PROGRAM NCI
VAR
  bInit                     : BOOL;
  eInit                     : E_PROGRESS;

  nChn,
  nChnInit,
  nAxis,
  nAxisInit                 : UINT;

  stMsg                     : ST_Message;

END_VAR

//-----------------------------------------------------------------------------------------------------------------
// check if compiler define is present [PLC_STATE_DRIVE/CompilerDefines/Manual: NCI]
// see PLC_CONSTANT for conditional pragma
//-----------------------------------------------------------------------------------------------------------------
IF NOT PLC_CONSTANT.NCI_ACTIVE THEN eInit   := E_PROGRESS.PROGRESS_NOT_EXIST; RETURN; END_IF
//-----------------------------------------------------------------------------------------------------------------
//-----------------------------------------------------------------------------------------------------------------
// check for MAIN.eInit
//-----------------------------------------------------------------------------------------------------------------
IF NOT (MAIN.eInit = E_PROGRESS.PROGRESS_DONE) THEN eInit   := E_PROGRESS.PROGRESS_INVALID; RETURN; END_IF
//-----------------------------------------------------------------------------------------------------------------
//-----------------------------------------------------------------------------------------------------------------
// /assign dataflow
//-----------------------------------------------------------------------------------------------------------------
FOR nChn := 1 TO MAX_NCI_CH
DO
  // NCI axis configuration --> NC AxisId used
  GVL_NCI.NciCtrl[nChn].ItfChannel.CfgAxes          := ADR(GVL_NCI.AxisConfig[nChn]);

  // R Parameter properties
  GVL_NCI.NciCtrl[nChn].ItfChannel.R_ParameterRead  := ADR(GVL_NCI.R_ParameterRead[nChn]);
  GVL_NCI.NciCtrl[nChn].ItfChannel.R_ParameterWrite := ADR(GVL_NCI.R_ParameterWrite[nChn]);

  // ProgName for channel
  GVL_NCI.NciCtrl[nChn].ItfChannel.Prog             := GVL_NCI.ChannelCtrl[nChn].sProgramName;

  // check REAL value to avoid exception
  IF NOT IsFinite(F_Real(GVL_NCI.ChannelCtrl[nChn].rOverride))
  THEN
    GVL_NCI.NciCtrl[nChn].ItfChannel.Override       := 0.0;
  ELSE
    GVL_NCI.NciCtrl[nChn].ItfChannel.Override       := GVL_NCI.ChannelCtrl[nChn].rOverride;
  END_IF

  // command and state structure assignement
  GVL_NCI.NciCtrl[nChn].ChnCtrl                     := ADR(GVL_NCI.ChannelCtrl[nChn]);
  GVL_NCI.NciCtrl[nChn].ChnState                    := ADR(GVL_NCI.ChannelState[nChn]);
END_FOR
//-----------------------------------------------------------------------------------------------------------------
// assign dataflow/
//-----------------------------------------------------------------------------------------------------------------
//-----------------------------------------------------------------------------------------------------------------
// /INIT
//-----------------------------------------------------------------------------------------------------------------
IF NOT bInit
THEN
  CASE eInit
  OF
    E_PROGRESS.PROGRESS_INVALID,
    E_PROGRESS.PROGRESS_DONE:
      FOR nChn := 1 TO MAX_NCI_CH
      DO
        GVL_MSG.MessageLevelNciChn[nChn]            := E_MessageType.eMessageVerbose;//GVL_MSG.MessageLevel;
      END_FOR
      nChnInit                                      := 1;
      eInit                                         := E_PROGRESS.PROGRESS_INIT;
    //-----------------------------------------------------------------------------
    //-----------------------------------------------------------------------------
    E_PROGRESS.PROGRESS_INIT:
      stMsg.eType                                   := E_MessageType.eMessageInfo;
      stMsg.eDevice                                 := e_Device.Device_Nci;
      stMsg.eSubdevice                              := e_SubDevice.MainInit;
      stMsg.iErrorNumber                            := MAX_AXIS;
      stMsg.sText                                   := concat('NCI.eInit: ', TO_STRING(eInit));
      f_MessageSet(stMsg);                          

      eInit                                         := E_PROGRESS.PROGRESS_BUSY;
    //-----------------------------------------------------------------------------
    //-----------------------------------------------------------------------------
    E_PROGRESS.PROGRESS_BUSY:
      eInit                                         := E_PROGRESS.PROGRESS_PREPARE;
    //-----------------------------------------------------------------------------
    //-----------------------------------------------------------------------------
    E_PROGRESS.PROGRESS_PREPARE:
      stMsg.eType                                   := E_MessageType.eMessageVerbose;
      stMsg.eDevice                                 := e_Device.Device_Nci;
      stMsg.eSubdevice                              := e_SubDevice.NciStartUp;
      stMsg.iErrorNumber                            := nChnInit;
      stMsg.sText                                   := concat('nChnInit: ', TO_STRING(nChnInit));

      IF (GVL_MSG.MessageLevelNciChn[nChnInit] = E_MessageType.eMessageVerbose)
      THEN
        f_MessageSet(stMsg);
      END_IF

      GVL_NCI.ChannelCtrl[nChnInit].eCmd            := E_NCI_CTRL.NULL;
      eInit                                         := E_PROGRESS.PROGRESS_STARTUP;
    //-----------------------------------------------------------------------------
    //-----------------------------------------------------------------------------
    E_PROGRESS.PROGRESS_STARTUP:
      GVL_NCI.ChannelCtrl[nChnInit].eCmd            := E_NCI_CTRL.INIT;

      IF (GVL_NCI.ChannelState[nChnInit].eState = E_NCI_STATE.INIT + E_PROGRESS.PROGRESS_ERROR)
      THEN
        eInit                                       := E_PROGRESS.PROGRESS_ERROR;

        stMsg.eType                                 := E_MessageType.eMessageError;
        stMsg.eDevice                               := e_Device.Device_Nci;
        stMsg.eSubdevice                            := e_SubDevice.NciStartUp;
        stMsg.iErrorNumber                          := nChnInit;
        stMsg.sText                                 := concat('NCI.eInit ERROR at Index: ', TO_STRING(nChnInit));
        f_MessageSet(stMsg);

      ELSIF (GVL_NCI.ChannelState[nChnInit].eState = E_NCI_STATE.INIT + E_PROGRESS.PROGRESS_DONE)
      THEN
        eInit                                       := E_PROGRESS.PROGRESS_CHECK;
      END_IF
    //-----------------------------------------------------------------------------
    //-----------------------------------------------------------------------------
    E_PROGRESS.PROGRESS_CHECK:
      IF (nChnInit > PLC_CONSTANT.MAX_NCI_CH-1)
      THEN
        bInit                                       := TRUE;
        eInit                                       := E_PROGRESS.PROGRESS_DONE;

        stMsg.eType                                 := E_MessageType.eMessageInfo;
        stMsg.eDevice                               := e_Device.Device_Nci;
        stMsg.eSubdevice                            := e_SubDevice.NciStartUp;
        stMsg.iErrorNumber                          := MAX_NCI_CH;
        stMsg.sText                                 := concat('NCI.eInit: ', TO_STRING(eInit));
        f_MessageSet(stMsg);

        FOR nChn := 1 TO MAX_NCI_CH
        DO
          GVL_MSG.MessageLevelNciChn[nChn]          := GVL_MSG.MessageLevel;
        END_FOR

      ELSE
        nChnInit                                    := nChnInit + 1;
        eInit                                       := E_PROGRESS.PROGRESS_PREPARE;
      END_IF
  END_CASE
END_IF
//-----------------------------------------------------------------------------------------------------------------
// INIT/
//-----------------------------------------------------------------------------------------------------------------
//-----------------------------------------------------------------------------------------------------------------
//-----------------------------------------------------------------------------------------------------------------
// /CYCLE
//-----------------------------------------------------------------------------------------------------------------
FOR nChn := 1 TO MAX_NCI_CH
DO
  // call nci channel controller
  GVL_NCI.NciCtrl[nChn].Cycle();

  GVL_NCI.ProgramNameActive[nChn]                   := GVL_NCI.NciCtrl[nChn].ItfChannel.GetLoadedProg();
  GVL_NCI.ChannelState[nChn].sProgramNameActive     := GVL_NCI.ProgramNameActive[nChn];
  GVL_NCI.NciCtrl[nChn].M_FunctionScope             := ADR(GVL_NCI.M_FunctionCyclic[nChn]);
END_FOR
//-----------------------------------------------------------------------------------------------------------------
// CYCLE/
//-----------------------------------------------------------------------------------------------------------------
//-----------------------------------------------------------------------------------------------------------------

END_PROGRAM

(* stored: Version 1.1.0.1, ProductVersion 3.1.4026.18
   POU NCI: Id {da86f3fe-4721-09d7-2e2d-987f1b92458d}, SpecialFunc None *)
